(* CODESYS project 3.project

Project tree, tasks and I/O mapping:
  Device : CODESYS Control Win V3, 3S - Smart Software Solutions GmbH, order no. 305021, version 3.5.11.30
    application Application
      libraries: Standard, * (System)
      task MainTask (cyclic, interval t#20ms, priority 1) calls PLC_PRG
      program PLC_PRG [LD]
*)

// Device/Application/PLC_PRG
PROGRAM PLC_PRG
VAR
	BT1: BOOL;
	B1: BOOL;
	PT1: BOOL;
	L1: BOOL;
END_VAR

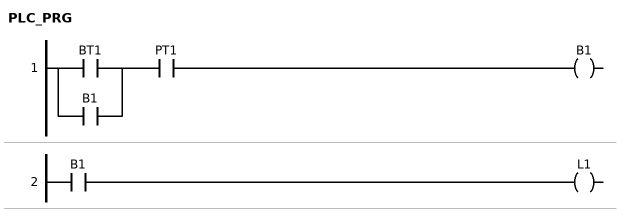
// NETWORK 1
B1 := (BT1 OR B1) AND PT1;

// NETWORK 2
L1 := B1;

END_PROGRAM
